(* PLC project Senza_nome, Sconosciuto Senza_nome 1 *)
(* stored: creationDateTime 2020-04-07T12:21:31, modificationDateTime 2020-04-07T15:51:19 *)

PROGRAM main_trapano
  VAR
    p : BOOL := 0;  (* pulsante di avvio *)
    a : BOOL := 0;  (* finecorsa alto *)
    m : BOOL := 0;  (* media corsa *)
    b : BOOL := 0;  (* finecorsa basso *)
    x : BOOL := 0;  (* sensore altezza pezzo *)
    y : BOOL := 0;  (* sensore presenza pezzo *)
    UP : BOOL := 0;  (* comando salita del trapano *)
    DWN : BOOL := 0;  (* comando discesa del trapano *)
    ROT : BOOL := 0;  (* comando rotazione del trapano *)
    OIL : BOOL := 0;  (* comando pompa olio *)
  END_VAR

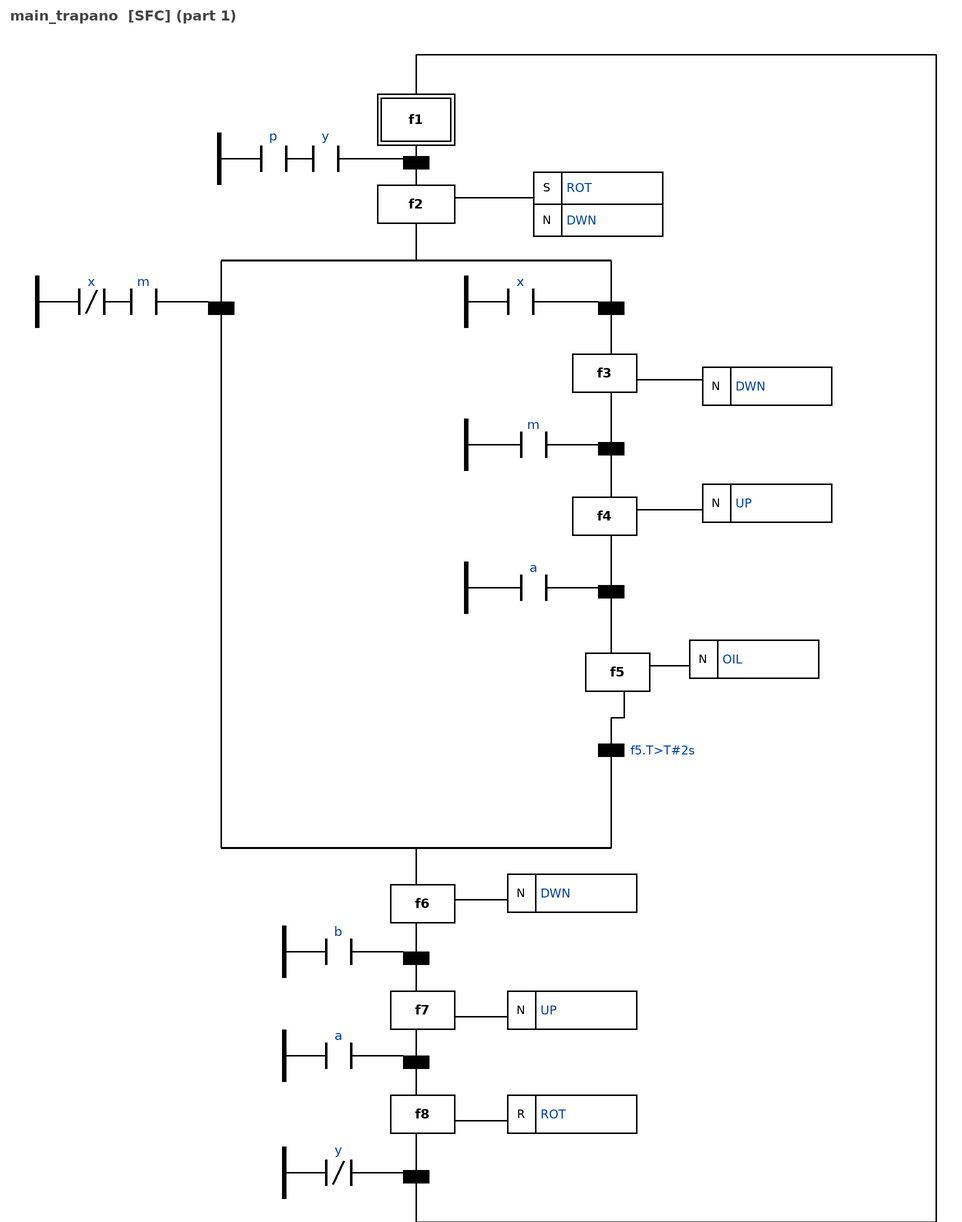
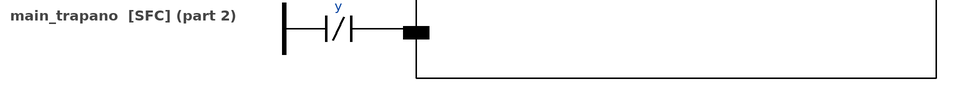
INITIAL_STEP f1:
END_STEP
TRANSITION FROM f1 TO f2
  := p AND y;
END_TRANSITION
STEP f2:
  ROT(S);
  DWN(N);
END_STEP
TRANSITION FROM f2 TO f6
  := NOT x AND m;
END_TRANSITION
TRANSITION FROM f2 TO f3
  := x;
END_TRANSITION
STEP f3:
  DWN(N);
END_STEP
TRANSITION FROM f3 TO f4
  := m;
END_TRANSITION
STEP f4:
  UP(N);
END_STEP
TRANSITION FROM f4 TO f5
  := a;
END_TRANSITION
STEP f5:
  OIL(N);
END_STEP
TRANSITION FROM f5 TO f6
  := f5.T>T#2s;
END_TRANSITION
STEP f6:
  DWN(N);
END_STEP
TRANSITION FROM f6 TO f7
  := b;
END_TRANSITION
STEP f7:
  UP(N);
END_STEP
TRANSITION FROM f7 TO f8
  := a;
END_TRANSITION
STEP f8:
  ROT(R);
END_STEP
TRANSITION FROM f8 TO f1
  := NOT y;
END_TRANSITION
END_PROGRAM

CONFIGURATION Config0
  RESOURCE Res0 ON PLC
    TASK task0(INTERVAL := T#20ms, PRIORITY := 0);
    PROGRAM instance0 WITH task0 : main_trapano;
  END_RESOURCE
END_CONFIGURATION
